TYPE T_SA_CH_STATE :
STRUCT
	//
	// Channel State
	// Got with the ':CHAN#:STAT?' command
	//
	bACTIVELY_MOVING:			BOOL;
	bCLOSED_LOOP_ACTIVE:		BOOL;
	bCALIBRATING:				BOOL;
	bREFERENCING:				BOOL;
	bMOVE_DELAYED:				BOOL;
	bSENSOR_PRESENT:			BOOL;
	bIS_CALIBRATED:				BOOL;
	bIS_REFERENCED:				BOOL;
	bEND_STOP_REACHED:			BOOL;
	bRANGE_LIMIT_REACHED:		BOOL;
	bFOLLOWING_LIMIT_REACHED:	BOOL;
	bMOVEMENT_FAILED:			BOOL;
	bIS_STREAMING:				BOOL;
	bPOSITIONER_OVERLOAD:		BOOL;
	bOVER_TEMPERATURE:			BOOL;
	bREFERENCE_MARK:			BOOL;
	bIS_PHASED:					BOOL;
	bPOSITIONER_FAULT:			BOOL;
	bAMPLIFIER_ENABLED:			BOOL;
	bIN_POSITION:				BOOL;

	bERROR:						BOOL := TRUE;
	
END_STRUCT
END_TYPE

(* stored: Version 1.1.0.1, ProductVersion 3.1.4024.10
   DUT T_SA_CH_STATE: Id {f7cb5c28-c4ab-4099-a73f-0efc8430de4b} *)
